{attribute 'qualified_only'}
VAR_GLOBAL	
	B1 AT %I*: BOOL; 	// Linearantrieb Endlage links (Öffner)
	B2 AT %I*: BOOL;	// Linearantrieb Endlage rechts (Öffner)
	S1 AT %I*: BOOL;	// Taster (1) (Schliesser)
	S2 AT %I*: BOOL;	// Taster (0) (Öffner)
	S3 AT %I*: BOOL;	// Taster I (Schliesser)
	S4 AT %I*: BOOL;	// Taster II (Schliesser)
	S5 AT %I*: BOOL;	// Taster Pfeil auf (Schliesser)
	S6 AT %I*: BOOL;	// Taster Pfeil ab (Schliesser)
	S7 AT %I*: BOOL;	// Taster + (Schliesser)
	S8 AT %I*: BOOL;	// Taster - (Schliesser)
	S9 AT %I*: BOOL;	// Taster STOP (Öffner)
	S10 AT %I*: BOOL;	// Taster Not Halt (Öffner)
	S11 AT %I*: BOOL;	// Taster Not Halt (Schliesser)
END_VAR

(* stored: Version 1.1.0.1, ProductVersion 3.1.4024.4
   GVL SimDI: Id {c2d05302-d374-4f85-80dd-41006a3e3277} *)
